{attribute 'GeneratedUsingTerminal: AMP8000-0030-0103-0103'}
{attribute addProperty BoxType "AMP8000-0030-0103-0103"}
{attribute addProperty Id "Ch_A_Following_error_actual_valueAT %I*DINT4"}
{attribute addProperty CRC "2360407386"}
{attribute addProperty Size "4"}
TYPE Ch_A_PositionControl_Inputs_8CB0F55A EXTENDS InputBase_8311D824 :
STRUCT
	{attribute addProperty Name "Ch_A_Following_error_actual_value"}
	Ch_A_Following_error_actual_value AT %I* : DINT;
END_STRUCT
END_TYPE

(* stored: Version 1.2.0.0, ProductVersion 3.1.4024.9
   DUT Ch_A_PositionControl_Inputs_8CB0F55A: Id {546e5769-dc6f-4474-bc0d-e8e5d2043ed8} *)
